PROGRAM MAIN
VAR
	
END_VAR

ReadingFile();
WritingFile();

END_PROGRAM

(* stored: Version 1.1.0.1
   POU MAIN: Id {5547197e-a179-4f8d-b8af-d7f4da8b9cce}, SpecialFunc None *)
